FUNCTION_BLOCK iterator
VAR_INPUT
	increment	:	DINT;
END_VAR
VAR_OUTPUT
	out	:	DINT;
END_VAR
VAR
	value	:	DINT	:=0;
	lim	:	DINT :=1000;
END_VAR

IF value < lim THEN
	value := value + increment;
ELSE
	value:= 0;	
END_IF
out := value;

END_FUNCTION_BLOCK

(* stored: Version 1.1.0.1, ProductVersion 3.1.4020.12
   POU iterator: Id {5a0e109f-dcdc-4a60-b655-31e2199f7b5b}, SpecialFunc None *)
